{attribute 'GeneratedUsingTerminal: EP9214-0023-0019'}
{attribute addProperty BoxType "EP9214-0023-0019"}
{attribute addProperty Id "Output_UsAT %Q*BOOL1Output_UpAT %Q*BOOL1Reset_UsAT %Q*BOOL1Reset_UpAT %Q*BOOL1"}
{attribute addProperty CRC "2757342060"}
{attribute addProperty Size "4"}
TYPE DPO_Outputs_Channel_A459B36C :
STRUCT
	{attribute addProperty Name "Output_Us"}
	Output_Us AT %Q* : BOOL;
	{attribute addProperty Name "Output_Up"}
	Output_Up AT %Q* : BOOL;
	{attribute addProperty Name "Reset_Us"}
	Reset_Us AT %Q* : BOOL;
	{attribute addProperty Name "Reset_Up"}
	Reset_Up AT %Q* : BOOL;
END_STRUCT
END_TYPE

(* stored: Version 1.2.0.0, ProductVersion 3.1.4024.9
   DUT DPO_Outputs_Channel_A459B36C: Id {c8c11812-1753-4061-aea9-1e3ebbd35191} *)
